FUNCTION F_GetAdsPort : UINT
VAR
    TaskIndex : DINT;
END_VAR

TaskIndex := GETCURTASKINDEXEX();
IF TaskIndex > 0 THEN
    F_GetAdsPort := TwinCAT_SystemInfoVarList._AppInfo.AdsPort;
END_IF

END_FUNCTION

(* stored: Version 1.1.0.1, ProductVersion 3.1.4020.12
   POU F_GetAdsPort: Id {a059fd71-612b-08fd-32c9-6351c977dbb7}, SpecialFunc None *)
